{library PUBLIC}
(*  Function to leave a pallet in a specific station and position.  *)
FUNCTION_BLOCK GantryLeave
VAR_INPUT
	En: 				BOOL:=FALSE;			(* Set to true to start *)
	LeaveStation:		StationType;			(* Station number 1-4 *)
	LeavePosition:		PositionType;			(* Position number 1-9 *)
END_VAR
VAR_OUTPUT
	Done: 				BOOL:=FALSE;			(* If true, the command is transmitted ok, to reset set En to false *)
	Executing:			BOOL:=FALSE;			(* True while the command in transmitted *)
	Waiting:			BOOL:=FALSE;			(* True if the command is queued to be transmitted *)
	Error: 				BOOL := FALSE;			(* True if an error occured *)
	Progress:			INT:=0;					(* Function progress *)
END_VAR
VAR_IN_OUT
	Data: 				CommunicationData;		(* Common data structure to connect this function block to a specific Communicator block *)
END_VAR
VAR
	FunctionType: 		FUNCTION_TYPE;
	FunctionNumber: 	INT;
	ParameterDW:	DWORD;
	ParameterB:		BYTE;
	ParametersOK:	BOOL;

	fbRPC:				ASyncRPC;
END_VAR


FunctionType:=FUNCTION_TYPE.FUNCTION_TYPE_ASYNC_RPC;
FunctionNumber:=GANTRY_ASYNC_FUNCTION_NUMBER.GANTRY_ASYNC_FUNCTION_PL;
ParameterDW:=0;
ParameterB:=0;
ParametersOK:=FALSE;

IF En THEN
	IF LeaveStation<=4 AND LeaveStation>=1 THEN
		IF LeavePosition<=9 AND LeavePosition>=1 THEN
			ParametersOK:=TRUE;
			ParameterDW:=INT_TO_DWORD( (0*1000+0*100) + (LeaveStation*10+LeavePosition));
		END_IF
	END_IF
END_IF

fbRPC(EN:=En AND ParametersOK, Data:=Data, FunctionType:=FunctionType,FunctionNumber:=FunctionNumber, ParameterDW:=ParameterDW, ParameterB:=ParameterB);

Done:=fbRPC.Done;
Executing:=fbRPC.Executing;
Waiting:=fbRPC.Waiting;
Error:=fbRPC.Error OR (fbRPC.Done AND fbRPC.ReturnValue<0) OR NOT ParametersOK;
Progress:=fbRPC.Progress;

END_FUNCTION_BLOCK

(* stored: Version 1.1.0.1, ProductVersion 3.1.4024.2
   POU GantryLeave: Id {f119961e-41ad-46eb-8331-6c782a0e61c2}, SpecialFunc None *)
